{attribute 'qualified_only'}
VAR_GLOBAL
	gfbAlarmManagement			: FB_AlarmManagement;	// first: nested FB_Alarm.FB_init prepends onto ipAlarmHead
	gfbLogFile					: FB_LogFile;
	gfbEventListener			: FB_EventListenerExtV2; // other HMI than TE2000
	ipAlarmHead					: I_Alarm;	// singly linked list of all FB_Alarm instances
	gnCountAlarms				: UINT := 0;	// built-in and user FB_Alarm instances self-register in FB_init
	gbCountAlarmsMaxExceeded	: BOOL := FALSE;
	gbInterfaceNotAssigned		: BOOL := FALSE;
	
END_VAR

(* stored: Version 1.1.0.1, ProductVersion 3.1.4026.18
   GVL GVL_Diag: Id {7bf02ed6-ce4b-4a1a-a562-eb7ee03f0ff7} *)
